FUNCTION F_LogDebug : STRING;
VAR_INPUT
   Message : T_MaxString;
END_VAR

F_LogDebug :=
   F_Logger(
      E_LogSeverity.Debug,
      CONCAT('DEBUG ', Message)
   );

END_FUNCTION

(* stored: Version 1.1.0.1, ProductVersion 3.1.4026.12
   POU F_LogDebug: Id {b9fa666b-0a86-0238-0973-36dd6b8fc96b}, SpecialFunc None *)
